(* PLC project Practical Work One, Rexroth ctrlX PLC Engineering ctrlX PLC 1.16.1, author Cedric Lenoir *)
(* stored: creationDateTime 2024-05-24T15:21:21.1871668, version 0.0, modificationDateTime 2024-05-24T15:19:54.2132771, organization HEVS *)
(* First Test for Practical Work One *)

TYPE UA_DigitalInput_32 : STRUCT
  Input_0_0 : BOOL;
  Input_0_1 : BOOL;
  Input_0_2 : BOOL;
  Input_0_3 : BOOL;
  Input_0_4 : BOOL;
  Input_0_5 : BOOL;
  Input_0_6 : BOOL;
  Input_0_7 : BOOL;
  Input_1_0 : BOOL;
  Input_1_1 : BOOL;
  Input_1_2 : BOOL;
  Input_1_3 : BOOL;
  Input_1_4 : BOOL;
  Input_1_5 : BOOL;
  Input_1_6 : BOOL;
  Input_1_7 : BOOL;
  Input_2_0 : BOOL;
  Input_2_1 : BOOL;
  Input_2_2 : BOOL;
  Input_2_3 : BOOL;
  Input_2_4 : BOOL;
  Input_2_5 : BOOL;
  Input_2_6 : BOOL;
  Input_2_7 : BOOL;
  Input_3_0 : BOOL;
  Input_3_1 : BOOL;
  Input_3_2 : BOOL;
  Input_3_3 : BOOL;
  Input_3_4 : BOOL;
  Input_3_5 : BOOL;
  Input_3_6 : BOOL;
  Input_3_7 : BOOL;
END_STRUCT;
END_TYPE

TYPE UA_DigitalOutput_32 : STRUCT
  Output_0_0 : BOOL;
  Output_0_1 : BOOL;
  Output_0_2 : BOOL;
  Output_0_3 : BOOL;
  Output_0_4 : BOOL;
  Output_0_5 : BOOL;
  Output_0_6 : BOOL;
  Output_0_7 : BOOL;
  Output_1_0 : BOOL;
  Output_1_1 : BOOL;
  Output_1_2 : BOOL;
  Output_1_3 : BOOL;
  Output_1_4 : BOOL;
  Output_1_5 : BOOL;
  Output_1_6 : BOOL;
  Output_1_7 : BOOL;
  Output_2_0 : BOOL;
  Output_2_1 : BOOL;
  Output_2_2 : BOOL;
  Output_2_3 : BOOL;
  Output_2_4 : BOOL;
  Output_2_5 : BOOL;
  Output_2_6 : BOOL;
  Output_2_7 : BOOL;
  Output_3_0 : BOOL;
  Output_3_1 : BOOL;
  Output_3_2 : BOOL;
  Output_3_3 : BOOL;
  Output_3_4 : BOOL;
  Output_3_5 : BOOL;
  Output_3_6 : BOOL;
  Output_3_7 : BOOL;
END_STRUCT;
END_TYPE

TYPE UA_ButtonAndSignal : STRUCT
  In_Estop : BOOL;
  In_Reset : BOOL;
  In_Start : BOOL;
  In_Stop : BOOL;
  Out_Idle : BOOL;
  Out_Execute : BOOL;
  Out_Stopped : BOOL;
END_STRUCT;
END_TYPE

TYPE UA_O300_DL : STRUCT
  Value : WORD;
  BCD1 : BOOL;
  Q : BOOL;
  A : BOOL;
END_STRUCT;
END_TYPE

TYPE UA_O300_ZL : STRUCT
  BCD1 : BOOL;
  Q : BOOL;
  A : BOOL;
END_STRUCT;
END_TYPE

TYPE UA_U300_D50 : STRUCT
  Value : DWORD;
  Scale : SINT;
  SSC1 : BOOL;
  SSC2 : BOOL;
  Q : BOOL;
  A : BOOL;
  SSC4 : BOOL;
END_STRUCT;
END_TYPE

(* www.hevs.ch Institut Systemes Industriels Project: Projet No: PW Move Absolute Author: Cedric Lenoir Date: 2023 October 16 Summary: List of commands for MoveAbsolute *)
TYPE ST_PlcOpenFbs : STRUCT
  bEnableRemote : BOOL;  (* If TRUE, the FB are driven manually from the HMI *)
  bEnableReadStatus : BOOL;
  bEnableReadPosition : BOOL;
  bEnableReadVelocity : BOOL;
  bMoveAbs : BOOL;
  bStop : BOOL;
  bPowerOn : BOOL;
  bReset : BOOL;
  strGetAxisStatus : STRING;  (* From arAxisStatus_gb[1].Data.PLCopenState; Exist in Data Layer too, s=motion/axs/Axis_X/state/opstate/plcopen *)
END_STRUCT;
END_TYPE

TYPE UA_U300_P50 : STRUCT
  Value : DWORD;
  Scale : SINT;
  SSC1 : BOOL;
  SSC2 : BOOL;
  Q : BOOL;
  A : BOOL;
  SSC4 : BOOL;
END_STRUCT;
END_TYPE

TYPE UA_Schunk_mms : STRUCT
  Value : WORD;
END_STRUCT;
END_TYPE

TYPE UA_Balluf_bcm0002 : STRUCT
  Data_1 : REAL;
  Data_2 : REAL;
  Data_3 : REAL;
  Temperature : REAL;
  Status : DWORD;
END_STRUCT;
END_TYPE

TYPE UA_Festo : STRUCT
  SetOut : BOOL;
END_STRUCT;
END_TYPE

TYPE UA_AnalogIn : STRUCT
  IW_04 : WORD;
  IW_06 : WORD;
  IW_08 : WORD;
  IW_10 : WORD;
  IW_12 : WORD;
  IW_14 : WORD;
  IW_16 : WORD;
  IW_18 : WORD;
END_STRUCT;
END_TYPE

TYPE UA_AnalogOut : STRUCT
  QW_04 : WORD;
  QW_06 : WORD;
  QW_08 : WORD;
  QW_10 : WORD;
END_STRUCT;
END_TYPE

TYPE UA_AboxInterface : STRUCT
  uaButtonAndSignal : UA_ButtonAndSignal;
  uaAnalogIn : UA_AnalogIn;
  uaAnalogOut : UA_AnalogOut;
  uaDigitalIn : UA_DigitalInput_32;
  uaDigitalOut : UA_DigitalOutput_32;
  uaO300_DL_Optic : UA_O300_DL;
  uaO300_ZL_Optic : UA_O300_ZL;
  uaU300_D50_Sound : UA_U300_D50;
  uaU300_P50_Sound : UA_U300_P50;
  uaSchunk : UA_Schunk_mms;
  uaSchunkGripper : UA_Festo;
  uaAccelerometer : UA_Balluf_bcm0002;
END_STRUCT;
END_TYPE

(* www.hevs.ch Institut Systemes Industriels Project: Projet No: PW Move Absolute Author: Cedric Lenoir Date: 2023 October 16 Summary: List of dynamic parameters for Move Absolute *)
TYPE ST_SetMotionParam : STRUCT
  rPosition_mm : LREAL;
  rVeloctiy_mm_s : LREAL;
  rAcceleration_mm_s2 : LREAL;
  rDeceleration_mm_s2 : LREAL;
  rJerk_mm_s3 : LREAL;
END_STRUCT;
END_TYPE

(* www.hevs.ch Institut Systemes Industriels Project: Projet No: PW Move Absolute Author: Cedric Lenoir Date: 2023 October 16 Summary: State Machine Info *)
TYPE ST_StateMachineInfo : STRUCT
  diState : DINT;
  eState : E_ExecuteCornerP5;
  strState : STRING;
END_STRUCT;
END_TYPE

{attribute 'qualified_only'}
{attribute 'strict'}
TYPE E_PackStates : (NotActive := 999, Aborted := 10, Clearing := 20, Stopped := 30, Resetting := 40, Idle := 50, Starting := 60, Stopping := 70, Aborting := 80, Execute := 90, Holding := 100, Held := 110, Unholding := 120, Suspending := 200, Suspended := 210, Unsuspending := 220, Completing := 300, Complete := 310) DINT;
END_TYPE

TYPE ST_PackState : STRUCT
  Aborted : BOOL;
  Clearing : BOOL;
  Stopped : BOOL;
  Resetting : BOOL;
  Idle : BOOL;
  Starting : BOOL;
  Stopping : BOOL;
  Aborting : BOOL;
  Execute : BOOL;
  Holding : BOOL;  (* Held Loop *)
  Held : BOOL;
  Unholding : BOOL;
  Suspending : BOOL;  (* Suspended Loop *)
  Suspended : BOOL;
  Unsuspending : BOOL;
  Completing : BOOL;  (* Complete Loop *)
  Complete : BOOL;
END_STRUCT;
END_TYPE

{attribute 'qualified_only'}
{attribute 'strict'}
TYPE E_Clearing : (eIdle := 99, eX_ErrorStop := 110, eX_Disabled := 120, eX_Enabled := 130, eY_ErrorStop := 210, eY_Disabled := 220, eY_Enabled := 230, eZ_ErrorStop := 310, eZ_Disabled := 320, eZ_Enabled := 330);
END_TYPE

{attribute 'qualified_only'}
{attribute 'strict'}
TYPE E_Stopping : (Idle := 99);
END_TYPE

{attribute 'qualified_only'}
{attribute 'strict'}
TYPE E_Resetting : (Idle := 99, eGripperSetOpen := 10, eGripperIsOpen := 20, eMotionInit_Z := 110, eMotionInitDone_Z := 120);
END_TYPE

{attribute 'qualified_only'}
{attribute 'strict'}
TYPE E_Starting : (Idle := 99, eMotionStarting := 10, eMotionStartingDone := 20);
END_TYPE

{attribute 'qualified_only'}
{attribute 'strict'}
TYPE E_InOpGripper : (IsIdle := 999, IsOpen := 10, IsClosed := 20, PartPresent := 30);
END_TYPE

TYPE ST_TestFbGripperHmi : STRUCT
  executeOpenDone : BOOL;
  executeCloseDone : BOOL;
  gripperStateClosed : BOOL;
  gripperStateOpen : BOOL;
  gripperStatePartPresent : BOOL;
  gripperStateError : BOOL;
  gripperStateInOp : BOOL;
END_STRUCT;
END_TYPE

{attribute 'qualified_only'}
{attribute 'strict'}
TYPE E_Aborting : (Idle := 99, Disabled := 1, ErrorStop := 2);
END_TYPE

TYPE ST_RemoteCyclicSetPosition : STRUCT
  in : ST_RemoteCyclicSetPositionIn;  (* Commands for program *)
  out : ST_RemoteCyclicSetPositionOut;  (* Status for program *)
END_STRUCT;
END_TYPE

TYPE ST_RemoteCyclicSetPositionIn : STRUCT
  lrStartPosition : LREAL := 0;  (* Set start position / Start of profile position *)
  lrEndPosition : LREAL := 50;  (* Set end position / End of profile position *)
  udiCycleTimeMultiplier : UDINT := 1000;  (* Cycle Time Multiplier, default is 1000 for 1000 ms *)
  bActivateCoupling : BOOL;  (* Activate coupling, when TRUE, axis position is set by fbGenerateProfile with 5th order polynomial *)
  bStartForward : BOOL;  (* Start polynomial profile forward *)
  lrProfileSetPosition : LREAL;  (* Set Position from Profile generator *)
END_STRUCT;
END_TYPE

TYPE ST_RemoteCyclicSetPositionOut : STRUCT
  bInitDone : BOOL;  (* Init done, ready for cyclic motion *)
  bError : BOOL;  (* There is an error *)
  bFwdDone : BOOL;  (* End of cyclic profile Forward *)
END_STRUCT;
END_TYPE

TYPE ST_Corner : STRUCT
  X : ST_SetMotionParam;
  Y : ST_SetMotionParam;
  Z : ST_SetMotionParam;
END_STRUCT;
END_TYPE

{attribute 'qualified_only'}
{attribute 'strict'}
TYPE E_InOperationDoneBase : (Idle := 999, Init := 10, InOp := 20, Error := 30, Done := 40);
END_TYPE

{attribute 'qualified_only'}
{attribute 'strict'}
TYPE E_ExecuteDone : (Idle := 999, Init := 10, InOp := 20, Done := 30, Error := 40);
END_TYPE

{attribute 'qualified_only'}
{attribute 'strict'}
TYPE E_InOperationBase : (Idle := 999, Init := 10, InOp := 20, Error := 30);
END_TYPE

{attribute 'qualified_only'}
{attribute 'strict'}
TYPE E_SubActiveP5 : (StartPointOut := 999, Running := 10, EndOfProfile := 20);
END_TYPE

(* www.hevs.ch Institut Systemes Industriels Project: Projet No: PW Move Absolute Author: Cedric Lenoir Date: 2024 April 02 Summary: Template of a program using PLCopen on partial Pack State Use a Cyclic Setpoint for motion in Pack Execute. *)
PROGRAM PRG_CyclicSetPoint
  VAR
    fbGripperState : FB_GripperState;  (* ********************************************************************************************************************* YOUR VARIABLES HERE ********************************************************************************************************************* *)
    fbOpenGripper : FB_OpenGripper;
    fbCloseGripper : FB_CloseGripper;
    uliCount : ULINT;
    bInitDone : BOOL;
    fbPackStates : FB_PackStates;  (* Pack Partial state machine *)
    eAborting : E_Aborting;
    eClearing : E_Clearing;
    eResetting : E_Resetting;
    eStarting : E_Starting;
    eStopping : E_Stopping;
    stStateMachineInfo : ST_StateMachineInfo;  (* State machine info for Execute *)
    stPlcOpenFbs : ST_PlcOpenFbs;  (* List of Structures *)
    stSetParam_X : ST_SetMotionParam := (rVeloctiy_mm_s := 2000, rAcceleration_mm_s2 := 1000, rDeceleration_mm_s2 := 1000, rJerk_mm_s3 := 1);
    stSetParam_Z : ST_SetMotionParam := (rVeloctiy_mm_s := 2000, rAcceleration_mm_s2 := 1000, rDeceleration_mm_s2 := 1000, rJerk_mm_s3 := 1);
    stCornerOne : ST_Corner := (X := (rVeloctiy_mm_s := 2000, rAcceleration_mm_s2 := 1000, rDeceleration_mm_s2 := 1000, rJerk_mm_s3 := 1), Y := (rVeloctiy_mm_s := 2000, rAcceleration_mm_s2 := 1000, rDeceleration_mm_s2 := 1000, rJerk_mm_s3 := 1), Z := (rVeloctiy_mm_s := 2000, rAcceleration_mm_s2 := 1000, rDeceleration_mm_s2 := 1000, rJerk_mm_s3 := 1));
    stCornerTwo : ST_Corner := (X := (rPosition_mm := 50, rVeloctiy_mm_s := 2000, rAcceleration_mm_s2 := 1000, rDeceleration_mm_s2 := 1000, rJerk_mm_s3 := 1), Y := (rVeloctiy_mm_s := 2000, rAcceleration_mm_s2 := 1000, rDeceleration_mm_s2 := 1000, rJerk_mm_s3 := 1), Z := (rVeloctiy_mm_s := 2000, rAcceleration_mm_s2 := 1000, rDeceleration_mm_s2 := 1000, rJerk_mm_s3 := 1));
    mcReadActualPos_X : MC_ReadActualPosition;  (* List of Function Blocks *)
    mcReadStatus_X : MC_ReadStatus;
    mcPower_X : MC_Power;
    mcMoveAbs_X : MC_MoveAbsolute;
    mcStop_X : MC_Stop := (Deceleration := 1);
    mcReset_X : MC_Reset;
    fbGenerateProfile : FB_GenerateP5;  (* Second part of variables are used to generate a motion profile using 5th order polynomial. Details of polynomials can be experimented using a mlx Matlab file. *)
    mcCyclicSetPoint : MB_CyclicSetPoint;
    mcReadActualPos_Z : MC_ReadActualPosition;  (* Simply used to move Z axis Up in a secure position *)
    mcReadStatus_Z : MC_ReadStatus;
    mcPower_Z : MC_Power;
    mcMoveAbs_Z : MC_MoveAbsolute;
    mcStop_Z : MC_Stop := (Deceleration := 1);
    mcReset_Z : MC_Reset;
    stTestFbGripperHmi : ST_TestFbGripperHmi;  (* Check your FB on HMI *)
  END_VAR

                    ACT_BaseInit();


IF fbPackStates.state.Execute THEN
	fbPackStates.Execute_SC := FALSE;
	(*
		Execute State Machine.
	*)
	CASE stStateMachineInfo.eState OF
		E_ExecuteCornerP5.eIdle :
			stStateMachineInfo.strState := 'Idle';
			
			stSetParam_X.rPosition_mm := 0;
			stStateMachineInfo.eState := E_ExecuteCornerP5.eMoveToCornerOne;

		E_ExecuteCornerP5.eMoveToCornerOne :
			stStateMachineInfo.strState := 'Motion To Corner One';
			IF mcMoveAbs_X.Done THEN
				stStateMachineInfo.eState := E_ExecuteCornerP5.eMoveToCornerOneDone; 
			END_IF

		E_ExecuteCornerP5.eMoveToCornerOneDone :
			stStateMachineInfo.strState := 'Motion To Corner One Done';
			// Corner 2 is like Corner three
			stSetParam_X.rPosition_mm := stCornerTwo.X.rPosition_mm;
			// stStateMachineInfo.eState := E_ExecuteCornerP5.eMoveToCornerThree;
			IF fbGripperState.IsOpen THEN
				stStateMachineInfo.eState := E_ExecuteCornerP5.eMoveToCornerTwo;
			END_IF;
			
 		(* Motion with P5*)   
    	E_ExecuteCornerP5.eMoveToCornerTwo :
			stStateMachineInfo.strState := 'Motion To Corner Two with P5';
			// Reset P5 to actual position
			// GVL_CyclSetPoint.stRemote.in.lrStartPosition := mcReadActualPos_X.Position;
			// Start position should be THIS position
			GVL_CyclSetPoint.stRemote.in.lrEndPosition := mcReadActualPos_X.Position;
			stStateMachineInfo.eState := E_ExecuteCornerP5.eEnableP5;
			
		E_ExecuteCornerP5.eEnableP5 :
			stStateMachineInfo.strState := 'Enable / Reset P5';
			IF fbGenerateProfile.Done THEN
				stStateMachineInfo.eState := E_ExecuteCornerP5.eCyclicSetPoint;
				;
			END_IF
		
		E_ExecuteCornerP5.eCyclicSetPoint :
			stStateMachineInfo.strState := 'Set Cyclic Set Point';
			IF mcCyclicSetPoint.Active THEN
				GVL_CyclSetPoint.stRemote.in.lrStartPosition := mcReadActualPos_X.Position;
				GVL_CyclSetPoint.stRemote.in.lrEndPosition := stCornerTwo.X.rPosition_mm;
				stStateMachineInfo.eState := E_ExecuteCornerP5.eFollowP5;
			END_IF
		
		E_ExecuteCornerP5.eFollowP5 :
			stStateMachineInfo.strState := 'Follow P5';
			IF fbGenerateProfile.Done THEN
				stStateMachineInfo.eState := E_ExecuteCornerP5.eStopCyclic;
			END_IF
		
		E_ExecuteCornerP5.eStopCyclic :
			stStateMachineInfo.strState := 'Stop Cyclic';
			IF mcStop_X.Done THEN
				stStateMachineInfo.eState := E_ExecuteCornerP5.eStopDone;
			END_IF
		
		E_ExecuteCornerP5.eStopDone :
			stStateMachineInfo.strState := 'Stop Done';
			stStateMachineInfo.eState := E_ExecuteCornerP5.eMoveToCornerTwoDone;	
		
		E_ExecuteCornerP5.eMoveToCornerTwoDone :			
			stStateMachineInfo.strState := 'Move to Corner Two Done';
			// Return to One.
			stSetParam_X.rPosition_mm := stCornerOne.X.rPosition_mm;
			IF fbGripperState.IsClosed THEN
				stStateMachineInfo.eState := E_ExecuteCornerP5.eMoveToCornerOne;
			END_IF; 

		E_ExecuteCornerP5.eMoveToCornerThree :
			stStateMachineInfo.strState := 'Motion to Corner Three';
			IF mcMoveAbs_X.Done THEN
				stStateMachineInfo.eState := E_ExecuteCornerP5.eMoveToCornerThreeDone; 
			END_IF

		E_ExecuteCornerP5.eMoveToCornerThreeDone :
			stStateMachineInfo.strState := 'Motion to Corner Three Done'; 

			stSetParam_X.rPosition_mm := 0;
			stStateMachineInfo.eState := E_ExecuteCornerP5.eMoveToCornerOne;

	END_CASE
	;
ELSE
	stStateMachineInfo.strState := 'Idle';
	stStateMachineInfo.eState := E_ExecuteCornerP5.eIdle;
END_IF

(*
	Try with 
*)
mcCyclicSetPoint.Execute := (GVL_CyclSetPoint.stRemote.in.bActivateCoupling AND stPlcOpenFbs.bEnableRemote) OR
	                        (stStateMachineInfo.eState = E_ExecuteCornerP5.eCyclicSetPoint);
mcCyclicSetPoint.SetPoint := GVL_CyclSetPoint.stRemote.in.lrProfileSetPosition;
mcCyclicSetPoint(Axis := GVL_AxisDefines.X_Axis);

(*
    Call FB at the end of the Program
*)
fbGenerateProfile(Enable := fbPackStates.state.Execute,
				  StartForward := (GVL_CyclSetPoint.stRemote.in.bStartForward AND stPlcOpenFbs.bEnableRemote) OR
                                   (stStateMachineInfo.eState = E_ExecuteCornerP5.eEnableP5)                   OR
                                   (stStateMachineInfo.eState = E_ExecuteCornerP5.eFollowP5),
                  startPosition_mm := GVL_CyclSetPoint.stRemote.in.lrStartPosition,		   // Start to try with 0
                  endPosition_mm := GVL_CyclSetPoint.stRemote.in.lrEndPosition,			   // Start to try with 50	
                  udiCyclTime_ms := GVL_CyclSetPoint.MOTION_CYCLE_TIME_ms,
                  udiCycleTimeMult := GVL_CyclSetPoint.stRemote.in.udiCycleTimeMultiplier, // Could be a parameter latter when all is working
                  arGoToPos := GVL_CyclSetPoint.arGoToPosition,
                  lrSetPosition => GVL_CyclSetPoint.stRemote.in.lrProfileSetPosition,
                  Done => GVL_CyclSetPoint.stRemote.out.bFwdDone);

(**********************************************************************************************************************
    Get Execute state machine in a DINT format
**********************************************************************************************************************)
stStateMachineInfo.diState := stStateMachineInfo.eState;
	
(**********************************************************************************************************************
	Utility FBs for motion, Do not modify
**********************************************************************************************************************)
ACT_ForAxis_X();
// Action for Y axis if defined
ACT_ForAxis_Z();

ACT_ForGripper();
                  

ACTION ACT_ForAxis_X:
                        (**********************************************************************************************************************
	X Axis
**********************************************************************************************************************)
mcReadStatus_X(Axis := GVL_AxisDefines.X_Axis,
               Enable := stPlcOpenFbs.bEnableReadStatus);

mcReadActualPos_X(Axis := GVL_AxisDefines.X_Axis,
                  Enable := stPlcOpenFbs.bEnableReadPosition);

mcPower_X(Axis := GVL_AxisDefines.X_Axis,
        Enable := (stPlcOpenFbs.bPowerOn AND stPlcOpenFbs.bEnableRemote) OR
                   		NOT stPlcOpenFbs.bEnableRemote AND 
				   		NOT (fbPackStates.state.Aborting OR
                             fbPackStates.state.Aborted));

mcStop_X(Axis := GVL_AxisDefines.X_Axis,
         Execute := (stPlcOpenFbs.bStop AND stPlcOpenFbs.bEnableRemote) OR
                    (fbPackStates.state.Stopping)                       OR
                    (stStateMachineInfo.eState = E_ExecuteCornerP5.eStopCyclic));

mcReset_X(Axis := GVL_AxisDefines.X_Axis,
        Execute := (stPlcOpenFbs.bReset AND stPlcOpenFbs.bEnableRemote) OR
                    fbPackStates.state.Aborting);

mcMoveAbs_X(Axis := GVL_AxisDefines.X_Axis,
            Position := stSetParam_X.rPosition_mm,
            Velocity := stSetParam_X.rVeloctiy_mm_s,
            Acceleration := stSetParam_X.rAcceleration_mm_s2,
            Deceleration := stSetParam_X.rDeceleration_mm_s2,
            Jerk := stSetParam_X.rJerk_mm_s3,
            Execute := (stPlcOpenFbs.bMoveAbs AND stPlcOpenFbs.bEnableRemote)    	OR
					   (eStarting = E_Starting.eMotionStarting)                  	OR
                       (stStateMachineInfo.eState = E_ExecuteCornerP5.eMoveToCornerOne)	OR              
                       (stStateMachineInfo.eState = E_ExecuteCornerP5.eMoveToCornerThree));  
						  

                      
END_ACTION

ACTION ACT_ForAxis_Z:
                        (**********************************************************************************************************************
	Z Axis
**********************************************************************************************************************)
mcReadStatus_Z(Axis := GVL_AxisDefines.Z_Axis,
               Enable := stPlcOpenFbs.bEnableReadStatus);

mcReadActualPos_Z(Axis := GVL_AxisDefines.Z_Axis,
                  Enable := stPlcOpenFbs.bEnableReadPosition);

mcPower_Z(Axis := GVL_AxisDefines.Z_Axis,
        Enable := (stPlcOpenFbs.bPowerOn AND stPlcOpenFbs.bEnableRemote) OR
                   		NOT stPlcOpenFbs.bEnableRemote AND 
				   		NOT (fbPackStates.state.Aborting OR
                             fbPackStates.state.Aborted));

// Note that a stop without deceleration leads to an error!!
mcStop_Z(Axis := GVL_AxisDefines.Z_Axis,
         Execute := (stPlcOpenFbs.bStop AND stPlcOpenFbs.bEnableRemote) OR
                     fbPackStates.state.Stopping);

mcReset_Z(Axis := GVL_AxisDefines.Z_Axis,
         Execute := (stPlcOpenFbs.bReset AND stPlcOpenFbs.bEnableRemote) OR
                     fbPackStates.state.Aborting);
					 
mcMoveAbs_Z(Axis := GVL_AxisDefines.Z_Axis,
            Position := stSetParam_Z.rPosition_mm,
            Velocity := stSetParam_Z.rVeloctiy_mm_s,
            Acceleration := stSetParam_Z.rAcceleration_mm_s2,
            Deceleration := stSetParam_Z.rDeceleration_mm_s2,
            Jerk := stSetParam_Z.rJerk_mm_s3,
            Execute := (stPlcOpenFbs.bMoveAbs AND stPlcOpenFbs.bEnableRemote)    OR
                       (eResetting = E_Resetting.eMotionInit_Z));  
                      
END_ACTION

ACTION ACT_BaseInit:
                        (*
    Some inits independant of the Main State Machine
*)
IF NOT bInitDone THEN
	bInitDone := TRUE;
    stPlcOpenFbs.bEnableReadStatus := TRUE;
    stPlcOpenFbs.bEnableReadPosition := TRUE;
    stPlcOpenFbs.bEnableReadVelocity := TRUE;
	// Init values to compile them and send to OPC_UA
	stTestFbGripperHmi.gripperStateClosed := FALSE;
	stTestFbGripperHmi.gripperStateOpen := FALSE;
	stTestFbGripperHmi.gripperStatePartPresent := FALSE;
	stTestFbGripperHmi.gripperStateError := FALSE;
	stTestFbGripperHmi.gripperStateInOp := FALSE;
	stTestFbGripperHmi.executeOpenDone := FALSE;
	stTestFbGripperHmi.executeCloseDone := FALSE;
END_IF

(*
    Remote conditions
*)
IF stPlcOpenFbs.bEnableRemote THEN
    IF mcMoveAbs_X.Done THEN
        stPlcOpenFbs.bMoveAbs := FALSE;
    END_IF
    IF mcStop_X.Done THEN
        stPlcOpenFbs.bStop := FALSE;
        stPlcOpenFbs.bMoveAbs := FALSE;
    END_IF
END_IF

// If remote, pack states are disabled
fbPackStates.SoftEstop := mcReadStatus_X.ErrorStop;
fbPackStates(Enable := NOT stPlcOpenFbs.bEnableRemote,
			 remote := GVL_Abox.uaAboxInterface.uaButtonAndSignal);
			 
(*
	Basically, only Acting state are used, wait state are doing nothing
	But sometimes, we could need to do something.. see Aborted.
*)

IF fbPackStates.state.Aborting THEN
	fbPackStates.Aborting_SC := TRUE;
ELSE
	;
END_IF

IF fbPackStates.state.Clearing THEN
	CASE eClearing OF
	E_Clearing.eIdle :
		IF mcReadStatus_X.Standstill THEN
			eClearing := E_Clearing.eY_ErrorStop;
		ELSIF mcReadStatus_X.ErrorStop THEN
			eClearing := E_Clearing.eX_ErrorStop;
		ELSE
			eClearing := E_Clearing.eX_Disabled;
		END_IF
	
	E_Clearing.eX_ErrorStop :
		IF mcReadStatus_X.Standstill THEN
			eClearing := E_Clearing.eY_ErrorStop;
		ELSE
			eClearing := E_Clearing.eX_Disabled;
		END_IF
	
	E_Clearing.eX_Disabled  :
		IF mcReadStatus_X.Standstill THEN
			eClearing := E_Clearing.eY_ErrorStop;
		ELSIF mcReadStatus_X.ErrorStop THEN
			eClearing := E_Clearing.eX_ErrorStop;
		END_IF
	
	E_Clearing.eX_Enabled   :
		IF mcReadStatus_X.Standstill THEN
			eClearing := E_Clearing.eY_ErrorStop;
		ELSIF mcReadStatus_X.ErrorStop THEN
			eClearing := E_Clearing.eX_ErrorStop;
		ELSE
			eClearing := E_Clearing.eX_Disabled;
		END_IF	

	E_Clearing.eY_ErrorStop :
		// No Y axis
		eClearing := E_Clearing.eZ_ErrorStop;
	
	E_Clearing.eY_Disabled  :
		eClearing := E_Clearing.eZ_ErrorStop;
	
	E_Clearing.eY_Enabled   :
		eClearing := E_Clearing.eZ_ErrorStop;

	E_Clearing.eZ_ErrorStop :
		IF mcReadStatus_Z.Standstill THEN
			eClearing := E_Clearing.eZ_Enabled;
		ELSE
			eClearing := E_Clearing.eZ_Disabled;
		END_IF	
	
	E_Clearing.eZ_Disabled  :
		IF mcReadStatus_Z.Standstill THEN
			eClearing := E_Clearing.eZ_Enabled;
		ELSIF mcReadStatus_Z.ErrorStop THEN
			eClearing := E_Clearing.eZ_ErrorStop;
		END_IF
	
	E_Clearing.eZ_Enabled   :;
		
	END_CASE
	// Reset Gripper in case fbOpenGripper and fbCloseGripper not presentz
	// GripperIsOpen   := TRUE;
	// GripperIsClosed	:= TRUE;	
	IF (eClearing = E_Clearing.eZ_Enabled) THEN
		fbPackStates.Clearing_SC := TRUE;
	ELSE
		fbPackStates.Clearing_SC := FALSE;
	END_IF
ELSE
	eClearing := E_Clearing.eIdle;
END_IF

IF fbPackStates.state.Stopping THEN
	IF mcReadStatus_X.Standstill AND
       mcReadStatus_Z.Standstill THEN
		fbPackStates.Stopping_SC := TRUE;
	ELSE
		fbPackStates.Stopping_SC := FALSE;
	END_IF
ELSE
	;
END_IF

(**********************************************************************************************************************
    Resetting
**********************************************************************************************************************)
IF fbPackStates.state.Resetting THEN
	fbPackStates.Resetting_SC := FALSE;
	CASE eResetting OF
		E_Resetting.Idle :
            stSetParam_Z.rPosition_mm := 0;
			stSetParam_Z.rVeloctiy_mm_s := 2000;  
			eResetting := E_Resetting.eGripperSetOpen;
			
		E_Resetting.eGripperSetOpen :
			IF fbGripperState.IsOpen THEN
				eResetting := E_Resetting.eGripperIsOpen;
			END_IF
			
		E_Resetting.eGripperIsOpen :
			// No Condition
			eResetting := E_Resetting.eMotionInit_Z;			
			
		E_Resetting.eMotionInit_Z :
			IF mcMoveAbs_Z.Done THEN
				eResetting := E_Resetting.eMotionInitDone_Z; 
			END_IF

		E_Resetting.eMotionInitDone_Z :
			;;
	END_CASE
	 
	IF eResetting = E_Resetting.eMotionInitDone_Z THEN
		fbPackStates.Resetting_SC := TRUE;
	END_IF
ELSE
	eResetting := E_Resetting.Idle;
END_IF

(**********************************************************************************************************************
    Starting
**********************************************************************************************************************)
IF fbPackStates.state.Starting THEN
	fbPackStates.Starting_SC := FALSE;
	CASE eStarting OF
		E_Starting.Idle :
			// Starting at corner Two
            stSetParam_X.rPosition_mm := stCornerOne.X.rPosition_mm;
			stSetParam_X.rVeloctiy_mm_s := stCornerOne.X.rVeloctiy_mm_s;  
			eStarting := E_Starting.eMotionStarting;

		E_Starting.eMotionStarting :
			IF mcMoveAbs_X.Done THEN
				eStarting := E_Starting.eMotionStartingDone; 
			END_IF

		E_Starting.eMotionStartingDone :
			;
						
	END_CASE
	 
	IF (eStarting = E_Starting.eMotionStartingDone) THEN
		fbPackStates.Starting_SC := TRUE;
	END_IF
ELSE
	eStarting := E_Starting.Idle;
END_IF
                      
END_ACTION

ACTION ACT_ForGripper:
                        fbGripperState.Enable := (stPlcOpenFbs.bEnableRemote)        		OR
                   		 (NOT stPlcOpenFbs.bEnableRemote 		AND 
				   		  NOT (fbPackStates.state.Aborting OR
                               fbPackStates.state.Aborted)); 
fbGripperState(hw := GVL_Abox.uaAboxInterface.uaSchunk);

stTestFbGripperHmi.gripperStateClosed := fbGripperState.IsClosed;
stTestFbGripperHmi.gripperStateOpen := fbGripperState.IsOpen;
stTestFbGripperHmi.gripperStatePartPresent := fbGripperState.PartPresent;
stTestFbGripperHmi.gripperStateError := fbGripperState.Error;
stTestFbGripperHmi.gripperStateInOp := fbGripperState.InOperation;

fbOpenGripper.Execute := (stStateMachineInfo.eState = E_ExecuteCornerP5.eMoveToCornerOneDone) OR 
                         (eResetting = E_Resetting.eGripperSetOpen);

fbCloseGripper.Execute := (stStateMachineInfo.eState = E_ExecuteCornerP5.eMoveToCornerTwoDone);

fbOpenGripper(hwEV := GVL_Abox.uaAboxInterface.uaSchunkGripper,
	          hwSensor := GVL_Abox.uaAboxInterface.uaSchunk,
			  Done => stTestFbGripperHmi.executeOpenDone);
			  
fbCloseGripper(hwEV := GVL_Abox.uaAboxInterface.uaSchunkGripper,
	          hwSensor := GVL_Abox.uaAboxInterface.uaSchunk,
			  Done => stTestFbGripperHmi.executeCloseDone);
                      
END_ACTION
END_PROGRAM

PROGRAM PRG_MapBox
  VAR
    UA_ReadCounterFromStation : DINT;  (* Write from Siemens to ctrX Core Used to check if read is running *)
    UA_ButtonAndSignal_In_Estop : BOOL;
    UA_ButtonAndSignal_In_Reset : BOOL;
    UA_ButtonAndSignal_In_Start : BOOL;
    UA_ButtonAndSignal_In_Stop : BOOL;
    UA_Balluf_bcm0002_Data_1 : REAL;
    UA_Balluf_bcm0002_Data_2 : REAL;
    UA_Balluf_bcm0002_Data_3 : REAL;
    UA_Balluf_bcm0002_Temperature : REAL;
    UA_Balluf_bcm0002_Status : DWORD;
    UA_Festo_SetOut : BOOL;
    UA_O300_DL_Value : WORD;
    UA_O300_DL_BCD1 : BOOL;
    UA_O300_DL_Q : BOOL;
    UA_O300_DL_A : BOOL;
    UA_O300_ZL_BCD1 : BOOL;
    UA_O300_ZL_Q : BOOL;
    UA_O300_ZL_A : BOOL;
    UA_U300_D50_Value : DWORD;
    UA_U300_D50_Scale : SINT;
    UA_U300_D50_SSC1 : BOOL;
    UA_U300_D50_SSC2 : BOOL;
    UA_U300_D50_Q : BOOL;
    UA_U300_D50_A : BOOL;
    UA_U300_D50_SSC4 : BOOL;
    UA_U300_P50_Value : DWORD;
    UA_U300_P50_Scale : SINT;
    UA_U300_P50_SSC1 : BOOL;
    UA_U300_P50_SSC2 : BOOL;
    UA_U300_P50_Q : BOOL;
    UA_U300_P50_A : BOOL;
    UA_U300_P50_SSC4 : BOOL;
    UA_DigitalInput_32_Input_0_0 : BOOL;
    UA_DigitalInput_32_Input_0_1 : BOOL;
    UA_DigitalInput_32_Input_0_2 : BOOL;
    UA_DigitalInput_32_Input_0_3 : BOOL;
    UA_DigitalInput_32_Input_0_4 : BOOL;
    UA_DigitalInput_32_Input_0_5 : BOOL;
    UA_DigitalInput_32_Input_0_6 : BOOL;
    UA_DigitalInput_32_Input_0_7 : BOOL;
    UA_DigitalInput_32_Input_1_0 : BOOL;
    UA_DigitalInput_32_Input_1_1 : BOOL;
    UA_DigitalInput_32_Input_1_2 : BOOL;
    UA_DigitalInput_32_Input_1_3 : BOOL;
    UA_DigitalInput_32_Input_1_4 : BOOL;
    UA_DigitalInput_32_Input_1_5 : BOOL;
    UA_DigitalInput_32_Input_1_6 : BOOL;
    UA_DigitalInput_32_Input_1_7 : BOOL;
    UA_DigitalInput_32_Input_2_0 : BOOL;
    UA_DigitalInput_32_Input_2_1 : BOOL;
    UA_DigitalInput_32_Input_2_2 : BOOL;
    UA_DigitalInput_32_Input_2_3 : BOOL;
    UA_DigitalInput_32_Input_2_4 : BOOL;
    UA_DigitalInput_32_Input_2_5 : BOOL;
    UA_DigitalInput_32_Input_2_6 : BOOL;
    UA_DigitalInput_32_Input_2_7 : BOOL;
    UA_DigitalInput_32_Input_3_0 : BOOL;
    UA_DigitalInput_32_Input_3_1 : BOOL;
    UA_DigitalInput_32_Input_3_2 : BOOL;
    UA_DigitalInput_32_Input_3_3 : BOOL;
    UA_DigitalInput_32_Input_3_4 : BOOL;
    UA_DigitalInput_32_Input_3_5 : BOOL;
    UA_DigitalInput_32_Input_3_6 : BOOL;
    UA_DigitalInput_32_Input_3_7 : BOOL;
    UA_WriteCounterToStation : DINT;  (* Siemens Read from ctrX Core Used to check if write is running *)
    UA_ButtonAndSignal_Out_Idle : BOOL;
    UA_ButtonAndSignal_Out_Execute : BOOL;
    UA_ButtonAndSignal_Out_Stopped : BOOL;
    UA_Schunk_mms_Value : WORD;
    UA_DigitalOutput_32_Output_0_0 : BOOL;
    UA_DigitalOutput_32_Output_0_1 : BOOL;
    UA_DigitalOutput_32_Output_0_2 : BOOL;
    UA_DigitalOutput_32_Output_0_3 : BOOL;
    UA_DigitalOutput_32_Output_0_4 : BOOL;
    UA_DigitalOutput_32_Output_0_5 : BOOL;
    UA_DigitalOutput_32_Output_0_6 : BOOL;
    UA_DigitalOutput_32_Output_0_7 : BOOL;
    UA_DigitalOutput_32_Output_1_0 : BOOL;
    UA_DigitalOutput_32_Output_1_1 : BOOL;
    UA_DigitalOutput_32_Output_1_2 : BOOL;
    UA_DigitalOutput_32_Output_1_3 : BOOL;
    UA_DigitalOutput_32_Output_1_4 : BOOL;
    UA_DigitalOutput_32_Output_1_5 : BOOL;
    UA_DigitalOutput_32_Output_1_6 : BOOL;
    UA_DigitalOutput_32_Output_1_7 : BOOL;
    UA_DigitalOutput_32_Output_2_0 : BOOL;
    UA_DigitalOutput_32_Output_2_1 : BOOL;
    UA_DigitalOutput_32_Output_2_2 : BOOL;
    UA_DigitalOutput_32_Output_2_3 : BOOL;
    UA_DigitalOutput_32_Output_2_4 : BOOL;
    UA_DigitalOutput_32_Output_2_5 : BOOL;
    UA_DigitalOutput_32_Output_2_6 : BOOL;
    UA_DigitalOutput_32_Output_2_7 : BOOL;
    UA_DigitalOutput_32_Output_3_0 : BOOL;
    UA_DigitalOutput_32_Output_3_1 : BOOL;
    UA_DigitalOutput_32_Output_3_2 : BOOL;
    UA_DigitalOutput_32_Output_3_3 : BOOL;
    UA_DigitalOutput_32_Output_3_4 : BOOL;
    UA_DigitalOutput_32_Output_3_5 : BOOL;
    UA_DigitalOutput_32_Output_3_6 : BOOL;
    UA_DigitalOutput_32_Output_3_7 : BOOL;
  END_VAR

                        (*
        Values from Profinet Station
    *)
    
    // Get Value from Profinet Station with UA Client Write
	GVL_Abox.uaAboxInterface.uaButtonAndSignal.In_Estop     := UA_ButtonAndSignal_In_Estop;
	GVL_Abox.uaAboxInterface.uaButtonAndSignal.In_Reset     := UA_ButtonAndSignal_In_Reset;
	GVL_Abox.uaAboxInterface.uaButtonAndSignal.In_Start     := UA_ButtonAndSignal_In_Start;
	GVL_Abox.uaAboxInterface.uaButtonAndSignal.In_Stop      := UA_ButtonAndSignal_In_Stop;
    // Values from Balluff accelerometer
    GVL_Abox.uaAboxInterface.uaAccelerometer.Data_1         := UA_Balluf_bcm0002_Data_1;
    GVL_Abox.uaAboxInterface.uaAccelerometer.Data_2         := UA_Balluf_bcm0002_Data_1;
    GVL_Abox.uaAboxInterface.uaAccelerometer.Data_3         := UA_Balluf_bcm0002_Data_1;
    GVL_Abox.uaAboxInterface.uaAccelerometer.Status         := UA_Balluf_bcm0002_Status;
    GVL_Abox.uaAboxInterface.uaAccelerometer.Temperature    := UA_Balluf_bcm0002_Temperature;

    // Values from Baumer O300 DL
    GVL_Abox.uaAboxInterface.uaO300_DL_Optic.Value          := UA_O300_DL_Value;                
    GVL_Abox.uaAboxInterface.uaO300_DL_Optic.A              := UA_O300_DL_A;                
    GVL_Abox.uaAboxInterface.uaO300_DL_Optic.Q              := UA_O300_DL_Q;                
    GVL_Abox.uaAboxInterface.uaO300_DL_Optic.BCD1           := UA_O300_DL_BCD1;                

    // Values from Baumer O300 ZL                
    GVL_Abox.uaAboxInterface.uaO300_ZL_Optic.A              := UA_O300_ZL_A;                
    GVL_Abox.uaAboxInterface.uaO300_ZL_Optic.Q              := UA_O300_ZL_Q;                
    GVL_Abox.uaAboxInterface.uaO300_ZL_Optic.BCD1           := UA_O300_ZL_BCD1;                

    // Values from Baumer U300 D50
    GVL_Abox.uaAboxInterface.uaU300_D50_Sound.Value         := UA_U300_D50_Value;  
    GVL_Abox.uaAboxInterface.uaU300_D50_Sound.A             := UA_U300_D50_A;  
    GVL_Abox.uaAboxInterface.uaU300_D50_Sound.Q             := UA_U300_D50_Q;  
    GVL_Abox.uaAboxInterface.uaU300_D50_Sound.Scale         := UA_U300_D50_Scale;  
    GVL_Abox.uaAboxInterface.uaU300_D50_Sound.SSC1          := UA_U300_D50_SSC1;  
    GVL_Abox.uaAboxInterface.uaU300_D50_Sound.SSC2          := UA_U300_D50_SSC2;  
    GVL_Abox.uaAboxInterface.uaU300_D50_Sound.SSC4          := UA_U300_D50_SSC4;  
    
    // Values from Baumer U300 P50
    GVL_Abox.uaAboxInterface.uaU300_P50_Sound.Value         := UA_U300_P50_Value;  
    GVL_Abox.uaAboxInterface.uaU300_P50_Sound.A             := UA_U300_P50_A;  
    GVL_Abox.uaAboxInterface.uaU300_P50_Sound.Q             := UA_U300_P50_Q;  
    GVL_Abox.uaAboxInterface.uaU300_P50_Sound.Scale         := UA_U300_P50_Scale;  
    GVL_Abox.uaAboxInterface.uaU300_P50_Sound.SSC1          := UA_U300_P50_SSC1;  
    GVL_Abox.uaAboxInterface.uaU300_P50_Sound.SSC2          := UA_U300_P50_SSC2;  
    GVL_Abox.uaAboxInterface.uaU300_P50_Sound.SSC4          := UA_U300_P50_SSC4;  
    
    // Values from Gripper sensor
    GVL_Abox.uaAboxInterface.uaSchunk.Value                 := UA_Schunk_mms_Value;  
    
    // Get 32 Digital Input
    GVL_Abox.uaAboxInterface.uaDigitalIn.Input_0_0          := UA_DigitalInput_32_Input_0_0;
    GVL_Abox.uaAboxInterface.uaDigitalIn.Input_0_1          := UA_DigitalInput_32_Input_0_1;
    GVL_Abox.uaAboxInterface.uaDigitalIn.Input_0_2          := UA_DigitalInput_32_Input_0_2;
    GVL_Abox.uaAboxInterface.uaDigitalIn.Input_0_3          := UA_DigitalInput_32_Input_0_3;
    GVL_Abox.uaAboxInterface.uaDigitalIn.Input_0_4          := UA_DigitalInput_32_Input_0_4;
    GVL_Abox.uaAboxInterface.uaDigitalIn.Input_0_5          := UA_DigitalInput_32_Input_0_5;
    GVL_Abox.uaAboxInterface.uaDigitalIn.Input_0_6          := UA_DigitalInput_32_Input_0_6;
    GVL_Abox.uaAboxInterface.uaDigitalIn.Input_0_7          := UA_DigitalInput_32_Input_0_7;
    GVL_Abox.uaAboxInterface.uaDigitalIn.Input_1_0          := UA_DigitalInput_32_Input_1_0;
    GVL_Abox.uaAboxInterface.uaDigitalIn.Input_1_1          := UA_DigitalInput_32_Input_1_1;
    GVL_Abox.uaAboxInterface.uaDigitalIn.Input_1_2          := UA_DigitalInput_32_Input_1_2;
    GVL_Abox.uaAboxInterface.uaDigitalIn.Input_1_3          := UA_DigitalInput_32_Input_1_3;
    GVL_Abox.uaAboxInterface.uaDigitalIn.Input_1_4          := UA_DigitalInput_32_Input_1_4;
    GVL_Abox.uaAboxInterface.uaDigitalIn.Input_1_5          := UA_DigitalInput_32_Input_1_5;
    GVL_Abox.uaAboxInterface.uaDigitalIn.Input_1_6          := UA_DigitalInput_32_Input_1_6;
    GVL_Abox.uaAboxInterface.uaDigitalIn.Input_1_7          := UA_DigitalInput_32_Input_1_7;
    GVL_Abox.uaAboxInterface.uaDigitalIn.Input_2_0          := UA_DigitalInput_32_Input_2_0;
    GVL_Abox.uaAboxInterface.uaDigitalIn.Input_2_1          := UA_DigitalInput_32_Input_2_1;
    GVL_Abox.uaAboxInterface.uaDigitalIn.Input_2_2          := UA_DigitalInput_32_Input_2_2;
    GVL_Abox.uaAboxInterface.uaDigitalIn.Input_2_3          := UA_DigitalInput_32_Input_2_3;
    GVL_Abox.uaAboxInterface.uaDigitalIn.Input_2_4          := UA_DigitalInput_32_Input_2_4;
    GVL_Abox.uaAboxInterface.uaDigitalIn.Input_2_5          := UA_DigitalInput_32_Input_2_5;
    GVL_Abox.uaAboxInterface.uaDigitalIn.Input_2_6          := UA_DigitalInput_32_Input_2_6;
    GVL_Abox.uaAboxInterface.uaDigitalIn.Input_2_7          := UA_DigitalInput_32_Input_2_7;
    GVL_Abox.uaAboxInterface.uaDigitalIn.Input_3_0          := UA_DigitalInput_32_Input_3_0;
    GVL_Abox.uaAboxInterface.uaDigitalIn.Input_3_1          := UA_DigitalInput_32_Input_3_1;
    GVL_Abox.uaAboxInterface.uaDigitalIn.Input_3_2          := UA_DigitalInput_32_Input_3_2;
    GVL_Abox.uaAboxInterface.uaDigitalIn.Input_3_3          := UA_DigitalInput_32_Input_3_3;
    GVL_Abox.uaAboxInterface.uaDigitalIn.Input_3_4          := UA_DigitalInput_32_Input_3_4;
    GVL_Abox.uaAboxInterface.uaDigitalIn.Input_3_5          := UA_DigitalInput_32_Input_3_5;
    GVL_Abox.uaAboxInterface.uaDigitalIn.Input_3_6          := UA_DigitalInput_32_Input_3_6;
    GVL_Abox.uaAboxInterface.uaDigitalIn.Input_3_7          := UA_DigitalInput_32_Input_3_7;
    
    (*
        Values to Profinet Station
    *)
	UA_WriteCounterToStation := UA_WriteCounterToStation + 1;

    // Set Visual Signals
	UA_ButtonAndSignal_Out_Execute 	:= GVL_Abox.uaAboxInterface.uaButtonAndSignal.Out_Execute;
	UA_ButtonAndSignal_Out_Idle 	:= GVL_Abox.uaAboxInterface.uaButtonAndSignal.Out_Idle;
	UA_ButtonAndSignal_Out_Stopped	:= GVL_Abox.uaAboxInterface.uaButtonAndSignal.Out_Stopped;
    
    // Set Gripper value
    UA_Festo_SetOut                 := NOT GVL_Abox.uaAboxInterface.uaSchunkGripper.SetOut;
    
    // Set 32 digital outputs
    UA_DigitalOutput_32_Output_0_0  := GVL_Abox.uaAboxInterface.uaDigitalOut.Output_0_0;
    UA_DigitalOutput_32_Output_0_1  := GVL_Abox.uaAboxInterface.uaDigitalOut.Output_0_1;
    UA_DigitalOutput_32_Output_0_2  := GVL_Abox.uaAboxInterface.uaDigitalOut.Output_0_2;
    UA_DigitalOutput_32_Output_0_3  := GVL_Abox.uaAboxInterface.uaDigitalOut.Output_0_3;
    UA_DigitalOutput_32_Output_0_4  := GVL_Abox.uaAboxInterface.uaDigitalOut.Output_0_4;
    UA_DigitalOutput_32_Output_0_5  := GVL_Abox.uaAboxInterface.uaDigitalOut.Output_0_5;
    UA_DigitalOutput_32_Output_0_6  := GVL_Abox.uaAboxInterface.uaDigitalOut.Output_0_6;
    UA_DigitalOutput_32_Output_0_7  := GVL_Abox.uaAboxInterface.uaDigitalOut.Output_0_7;
    UA_DigitalOutput_32_Output_1_0  := GVL_Abox.uaAboxInterface.uaDigitalOut.Output_1_0;
    UA_DigitalOutput_32_Output_1_1  := GVL_Abox.uaAboxInterface.uaDigitalOut.Output_1_1;
    UA_DigitalOutput_32_Output_1_2  := GVL_Abox.uaAboxInterface.uaDigitalOut.Output_1_2;
    UA_DigitalOutput_32_Output_1_3  := GVL_Abox.uaAboxInterface.uaDigitalOut.Output_1_3;
    UA_DigitalOutput_32_Output_1_4  := GVL_Abox.uaAboxInterface.uaDigitalOut.Output_1_4;
    UA_DigitalOutput_32_Output_1_5  := GVL_Abox.uaAboxInterface.uaDigitalOut.Output_1_5;
    UA_DigitalOutput_32_Output_1_6  := GVL_Abox.uaAboxInterface.uaDigitalOut.Output_1_6;
    UA_DigitalOutput_32_Output_1_7  := GVL_Abox.uaAboxInterface.uaDigitalOut.Output_1_7;
    UA_DigitalOutput_32_Output_2_0  := GVL_Abox.uaAboxInterface.uaDigitalOut.Output_2_0;
    UA_DigitalOutput_32_Output_2_1  := GVL_Abox.uaAboxInterface.uaDigitalOut.Output_2_1;
    UA_DigitalOutput_32_Output_2_2  := GVL_Abox.uaAboxInterface.uaDigitalOut.Output_2_2;
    UA_DigitalOutput_32_Output_2_3  := GVL_Abox.uaAboxInterface.uaDigitalOut.Output_2_3;
    UA_DigitalOutput_32_Output_2_4  := GVL_Abox.uaAboxInterface.uaDigitalOut.Output_2_4;
    UA_DigitalOutput_32_Output_2_5  := GVL_Abox.uaAboxInterface.uaDigitalOut.Output_2_5;
    UA_DigitalOutput_32_Output_2_6  := GVL_Abox.uaAboxInterface.uaDigitalOut.Output_2_6;
    UA_DigitalOutput_32_Output_2_7  := GVL_Abox.uaAboxInterface.uaDigitalOut.Output_2_7;
    UA_DigitalOutput_32_Output_3_0  := GVL_Abox.uaAboxInterface.uaDigitalOut.Output_3_0;
    UA_DigitalOutput_32_Output_3_1  := GVL_Abox.uaAboxInterface.uaDigitalOut.Output_3_1;
    UA_DigitalOutput_32_Output_3_2  := GVL_Abox.uaAboxInterface.uaDigitalOut.Output_3_2;
    UA_DigitalOutput_32_Output_3_3  := GVL_Abox.uaAboxInterface.uaDigitalOut.Output_3_3;
    UA_DigitalOutput_32_Output_3_4  := GVL_Abox.uaAboxInterface.uaDigitalOut.Output_3_4;
    UA_DigitalOutput_32_Output_3_5  := GVL_Abox.uaAboxInterface.uaDigitalOut.Output_3_5;
    UA_DigitalOutput_32_Output_3_6  := GVL_Abox.uaAboxInterface.uaDigitalOut.Output_3_6;
    UA_DigitalOutput_32_Output_3_7  := GVL_Abox.uaAboxInterface.uaDigitalOut.Output_3_7;
    
PRG_CHECK_IO();
                  
END_PROGRAM

PROGRAM PRG_CHECK_IO
  VAR
    testButton_1 : BOOL;
    testButton_2 : BOOL;
    testButton_3 : BOOL;
    clignote : TON;
    changeMeSlow : BOOL;
    clignoteSlow : TON;
    changeMe : BOOL;
    NotResetTest : BOOL := TRUE;
  END_VAR

                    testButton_1 := GVL_Abox.uaAboxInterface.uaButtonAndSignal.In_Reset;
testButton_2 := GVL_Abox.uaAboxInterface.uaButtonAndSignal.In_Start;
testButton_3 := GVL_Abox.uaAboxInterface.uaButtonAndSignal.In_Stop;

IF GVL_Abox.uaAboxInterface.uaButtonAndSignal.In_Reset AND
   NotResetTest										   THEN
	NotResetTest := FALSE;
	
    GVL_Abox.uaAboxInterface.uaSchunkGripper.SetOut := FALSE;
    
    GVL_Abox.uaAboxInterface.uaButtonAndSignal.Out_Execute := FALSE;	
    GVL_Abox.uaAboxInterface.uaButtonAndSignal.Out_Idle := FALSE;	
    GVL_Abox.uaAboxInterface.uaButtonAndSignal.Out_Stopped := FALSE;	

    GVL_Abox.uaAboxInterface.uaDigitalOut.Output_0_0 := FALSE;
    GVL_Abox.uaAboxInterface.uaDigitalOut.Output_0_1 := FALSE;
    GVL_Abox.uaAboxInterface.uaDigitalOut.Output_0_2 := FALSE;
    GVL_Abox.uaAboxInterface.uaDigitalOut.Output_0_3 := FALSE;
    GVL_Abox.uaAboxInterface.uaDigitalOut.Output_0_4 := FALSE;
    GVL_Abox.uaAboxInterface.uaDigitalOut.Output_0_5 := FALSE;
    GVL_Abox.uaAboxInterface.uaDigitalOut.Output_0_6 := FALSE;
    GVL_Abox.uaAboxInterface.uaDigitalOut.Output_0_7 := FALSE;
    
    GVL_Abox.uaAboxInterface.uaDigitalOut.Output_1_0 := FALSE;
    GVL_Abox.uaAboxInterface.uaDigitalOut.Output_1_1 := FALSE;
    GVL_Abox.uaAboxInterface.uaDigitalOut.Output_1_2 := FALSE;
    GVL_Abox.uaAboxInterface.uaDigitalOut.Output_1_3 := FALSE;
    GVL_Abox.uaAboxInterface.uaDigitalOut.Output_1_4 := FALSE;
    GVL_Abox.uaAboxInterface.uaDigitalOut.Output_1_5 := FALSE;
    GVL_Abox.uaAboxInterface.uaDigitalOut.Output_1_6 := FALSE;
    GVL_Abox.uaAboxInterface.uaDigitalOut.Output_1_7 := FALSE;
    
    GVL_Abox.uaAboxInterface.uaDigitalOut.Output_2_0 := FALSE;
    GVL_Abox.uaAboxInterface.uaDigitalOut.Output_2_1 := FALSE;
    GVL_Abox.uaAboxInterface.uaDigitalOut.Output_2_2 := FALSE;
    GVL_Abox.uaAboxInterface.uaDigitalOut.Output_2_3 := FALSE;
    GVL_Abox.uaAboxInterface.uaDigitalOut.Output_2_4 := FALSE;
    GVL_Abox.uaAboxInterface.uaDigitalOut.Output_2_5 := FALSE;
    GVL_Abox.uaAboxInterface.uaDigitalOut.Output_2_6 := FALSE;
    GVL_Abox.uaAboxInterface.uaDigitalOut.Output_2_7 := FALSE;

    GVL_Abox.uaAboxInterface.uaDigitalOut.Output_3_0 := FALSE;
    GVL_Abox.uaAboxInterface.uaDigitalOut.Output_3_1 := FALSE;
    GVL_Abox.uaAboxInterface.uaDigitalOut.Output_3_2 := FALSE;
    GVL_Abox.uaAboxInterface.uaDigitalOut.Output_3_3 := FALSE;
    GVL_Abox.uaAboxInterface.uaDigitalOut.Output_3_4 := FALSE;
    GVL_Abox.uaAboxInterface.uaDigitalOut.Output_3_5 := FALSE;
    GVL_Abox.uaAboxInterface.uaDigitalOut.Output_3_6 := FALSE;
    GVL_Abox.uaAboxInterface.uaDigitalOut.Output_3_7 := FALSE;	
END_IF

IF GVL_Abox.uaAboxInterface.uaButtonAndSignal.In_Reset AND
   GVL_Abox.uaAboxInterface.uaButtonAndSignal.In_Start AND
   GVL_Abox.uaAboxInterface.uaButtonAndSignal.In_Stop  THEN
	NotResetTest := TRUE;
END_IF


IF NotResetTest THEN 
	
	// Quick Blink
	clignote(IN := changeMe,
			 PT := T#500MS);
			 
	IF clignote.Q THEN
		changeMe := FALSE;
	ELSE
		changeMe := TRUE;
	END_IF

	// Slow Blink
	clignoteSlow(IN := changeMeSlow,
			 	 PT := T#2500MS);
			 
	IF clignoteSlow.Q THEN
		changeMeSlow := FALSE;
	ELSE
		changeMeSlow := TRUE;
	END_IF
	
	IF (NOT GVL_Abox.uaAboxInterface.uaSchunkGripper.SetOut) AND clignoteSlow.Q THEN
		GVL_Abox.uaAboxInterface.uaSchunkGripper.SetOut := TRUE;
	ELSIF GVL_Abox.uaAboxInterface.uaSchunkGripper.SetOut AND clignoteSlow.Q THEN
		GVL_Abox.uaAboxInterface.uaSchunkGripper.SetOut := FALSE;
	END_IF
	
	IF (NOT GVL_Abox.uaAboxInterface.uaDigitalOut.Output_0_0) AND clignote.Q THEN
		GVL_Abox.uaAboxInterface.uaButtonAndSignal.Out_Execute := TRUE;	
		GVL_Abox.uaAboxInterface.uaButtonAndSignal.Out_Idle := TRUE;	
		GVL_Abox.uaAboxInterface.uaButtonAndSignal.Out_Stopped := TRUE;	
	
		GVL_Abox.uaAboxInterface.uaDigitalOut.Output_0_0 := TRUE;
		GVL_Abox.uaAboxInterface.uaDigitalOut.Output_0_1 := TRUE;
		GVL_Abox.uaAboxInterface.uaDigitalOut.Output_0_2 := TRUE;
		GVL_Abox.uaAboxInterface.uaDigitalOut.Output_0_3 := TRUE;
		GVL_Abox.uaAboxInterface.uaDigitalOut.Output_0_4 := TRUE;
		GVL_Abox.uaAboxInterface.uaDigitalOut.Output_0_5 := TRUE;
		GVL_Abox.uaAboxInterface.uaDigitalOut.Output_0_6 := TRUE;
		GVL_Abox.uaAboxInterface.uaDigitalOut.Output_0_7 := TRUE;
		
		GVL_Abox.uaAboxInterface.uaDigitalOut.Output_1_0 := TRUE;
		GVL_Abox.uaAboxInterface.uaDigitalOut.Output_1_1 := TRUE;
		GVL_Abox.uaAboxInterface.uaDigitalOut.Output_1_2 := TRUE;
		GVL_Abox.uaAboxInterface.uaDigitalOut.Output_1_3 := TRUE;
		GVL_Abox.uaAboxInterface.uaDigitalOut.Output_1_4 := TRUE;
		GVL_Abox.uaAboxInterface.uaDigitalOut.Output_1_5 := TRUE;
		GVL_Abox.uaAboxInterface.uaDigitalOut.Output_1_6 := TRUE;
		GVL_Abox.uaAboxInterface.uaDigitalOut.Output_1_7 := TRUE;
		
		GVL_Abox.uaAboxInterface.uaDigitalOut.Output_2_0 := TRUE;
		GVL_Abox.uaAboxInterface.uaDigitalOut.Output_2_1 := TRUE;
		GVL_Abox.uaAboxInterface.uaDigitalOut.Output_2_2 := TRUE;
		GVL_Abox.uaAboxInterface.uaDigitalOut.Output_2_3 := TRUE;
		GVL_Abox.uaAboxInterface.uaDigitalOut.Output_2_4 := TRUE;
		GVL_Abox.uaAboxInterface.uaDigitalOut.Output_2_5 := TRUE;
		GVL_Abox.uaAboxInterface.uaDigitalOut.Output_2_6 := TRUE;
		GVL_Abox.uaAboxInterface.uaDigitalOut.Output_2_7 := TRUE;

		GVL_Abox.uaAboxInterface.uaDigitalOut.Output_3_0 := TRUE;
		GVL_Abox.uaAboxInterface.uaDigitalOut.Output_3_1 := TRUE;
		GVL_Abox.uaAboxInterface.uaDigitalOut.Output_3_2 := TRUE;
		GVL_Abox.uaAboxInterface.uaDigitalOut.Output_3_3 := TRUE;
		GVL_Abox.uaAboxInterface.uaDigitalOut.Output_3_4 := TRUE;
		GVL_Abox.uaAboxInterface.uaDigitalOut.Output_3_5 := TRUE;
		GVL_Abox.uaAboxInterface.uaDigitalOut.Output_3_6 := TRUE;
		GVL_Abox.uaAboxInterface.uaDigitalOut.Output_3_7 := TRUE;
	ELSIF GVL_Abox.uaAboxInterface.uaDigitalOut.Output_0_0 AND clignote.Q THEN
		GVL_Abox.uaAboxInterface.uaButtonAndSignal.Out_Execute := FALSE;	
		GVL_Abox.uaAboxInterface.uaButtonAndSignal.Out_Idle := FALSE;	
		GVL_Abox.uaAboxInterface.uaButtonAndSignal.Out_Stopped := FALSE;	

		GVL_Abox.uaAboxInterface.uaDigitalOut.Output_0_0 := FALSE;
		GVL_Abox.uaAboxInterface.uaDigitalOut.Output_0_1 := FALSE;
		GVL_Abox.uaAboxInterface.uaDigitalOut.Output_0_2 := FALSE;
		GVL_Abox.uaAboxInterface.uaDigitalOut.Output_0_3 := FALSE;
		GVL_Abox.uaAboxInterface.uaDigitalOut.Output_0_4 := FALSE;
		GVL_Abox.uaAboxInterface.uaDigitalOut.Output_0_5 := FALSE;
		GVL_Abox.uaAboxInterface.uaDigitalOut.Output_0_6 := FALSE;
		GVL_Abox.uaAboxInterface.uaDigitalOut.Output_0_7 := FALSE;
		
		GVL_Abox.uaAboxInterface.uaDigitalOut.Output_1_0 := FALSE;
		GVL_Abox.uaAboxInterface.uaDigitalOut.Output_1_1 := FALSE;
		GVL_Abox.uaAboxInterface.uaDigitalOut.Output_1_2 := FALSE;
		GVL_Abox.uaAboxInterface.uaDigitalOut.Output_1_3 := FALSE;
		GVL_Abox.uaAboxInterface.uaDigitalOut.Output_1_4 := FALSE;
		GVL_Abox.uaAboxInterface.uaDigitalOut.Output_1_5 := FALSE;
		GVL_Abox.uaAboxInterface.uaDigitalOut.Output_1_6 := FALSE;
		GVL_Abox.uaAboxInterface.uaDigitalOut.Output_1_7 := FALSE;
		
		GVL_Abox.uaAboxInterface.uaDigitalOut.Output_2_0 := FALSE;
		GVL_Abox.uaAboxInterface.uaDigitalOut.Output_2_1 := FALSE;
		GVL_Abox.uaAboxInterface.uaDigitalOut.Output_2_2 := FALSE;
		GVL_Abox.uaAboxInterface.uaDigitalOut.Output_2_3 := FALSE;
		GVL_Abox.uaAboxInterface.uaDigitalOut.Output_2_4 := FALSE;
		GVL_Abox.uaAboxInterface.uaDigitalOut.Output_2_5 := FALSE;
		GVL_Abox.uaAboxInterface.uaDigitalOut.Output_2_6 := FALSE;
		GVL_Abox.uaAboxInterface.uaDigitalOut.Output_2_7 := FALSE;

		GVL_Abox.uaAboxInterface.uaDigitalOut.Output_3_0 := FALSE;
		GVL_Abox.uaAboxInterface.uaDigitalOut.Output_3_1 := FALSE;
		GVL_Abox.uaAboxInterface.uaDigitalOut.Output_3_2 := FALSE;
		GVL_Abox.uaAboxInterface.uaDigitalOut.Output_3_3 := FALSE;
		GVL_Abox.uaAboxInterface.uaDigitalOut.Output_3_4 := FALSE;
		GVL_Abox.uaAboxInterface.uaDigitalOut.Output_3_5 := FALSE;
		GVL_Abox.uaAboxInterface.uaDigitalOut.Output_3_6 := FALSE;
		GVL_Abox.uaAboxInterface.uaDigitalOut.Output_3_7 := FALSE;
	END_IF;
END_IF
                  
END_PROGRAM

FUNCTION_BLOCK FB_PackStates
  VAR_INPUT
    Enable : BOOL;
    SoftEstop : BOOL;
    Hold : BOOL := FALSE;
    Unhold : BOOL := FALSE;
    Clearing_SC : BOOL := TRUE;
    Stopping_SC : BOOL := TRUE;
    Aborting_SC : BOOL := TRUE;
    Resetting_SC : BOOL := TRUE;
    Starting_SC : BOOL := TRUE;
    Execute_SC : BOOL := FALSE;
    Holding_SC : BOOL := FALSE;
    Unholding_SC : BOOL := FALSE;
  END_VAR
  VAR_IN_OUT
    remote : UA_ButtonAndSignal;
  END_VAR
  VAR_OUTPUT
    state : ST_PackState;
    strState : STRING;
  END_VAR
  VAR
    initialized : BOOL;
    ePackStates : E_PackStates;
    rTrigStop : R_TRIG;
    rTrigStart : R_TRIG;
    rTrigReset : R_TRIG;
    clignote : TON;
    changeMe : BOOL;
  END_VAR

                    // 
//	Init
//
IF Enable THEN
	IF NOT initialized THEN
		// Init at Aborted when entering state machine.
		initialized := TRUE;
		ePackStates := E_PackStates.Aborted;
	END_IF;
ELSE
	ePackStates := E_PackStates.NotActive;
	initialized := FALSE;
END_IF

//
//	Manage Inputs
//
rTrigStop(CLK := remote.In_Stop);
rTrigStart(CLK := remote.In_Start);
rTrigReset(CLK := remote.In_Reset);

CASE ePackStates OF
	E_PackStates.NotActive	:
		strState := 'Not Active';
		;
	E_PackStates.Aborting 	:;
		strState := 'Aborting';
		IF Aborting_SC THEN
			ePackStates := E_PackStates.Aborted;
		END_IF
		
	E_PackStates.Aborted 	:
		strState := 'Aborted';
		IF rTrigReset.Q THEN
			ePackStates := E_PackStates.Clearing;
		END_IF
	
	E_PackStates.Clearing 	:
		strState := 'Clearing';
		// E-Stop Active Low
		IF NOT remote.In_Estop OR SoftEstop THEN
			ePackStates := E_PackStates.Aborting;
		ELSIF Clearing_SC THEN
			ePackStates := E_PackStates.Stopped;	
		END_IF

	E_PackStates.Stopped 	:
		strState := 'Stopped';
		// E-Stop Active Low
		IF NOT remote.In_Estop OR SoftEstop THEN
			ePackStates := E_PackStates.Aborting;
		ELSIF rTrigReset.Q THEN
			ePackStates := E_PackStates.Resetting;
		END_IF

	E_PackStates.Stopping 	:
		strState := 'Stopping';
		// E-Stop Active Low
		IF NOT remote.In_Estop OR SoftEstop THEN
			ePackStates := E_PackStates.Aborting;
		ELSIF Stopping_SC THEN
			ePackStates := E_PackStates.Stopped;
		END_IF

	E_PackStates.Resetting 	:
		strState := 'Resetting';
		// E-Stop Active Low
		IF NOT remote.In_Estop OR SoftEstop THEN
			ePackStates := E_PackStates.Aborting;
		ELSIF rTrigStop.Q THEN
			ePackStates := E_PackStates.Stopping;
		ELSIF Resetting_SC THEN
			ePackStates := E_PackStates.Idle;			
		END_IF

	E_PackStates.Idle 		:
		strState := 'Idle';
		// E-Stop Active Low
		IF NOT remote.In_Estop OR SoftEstop THEN
			ePackStates := E_PackStates.Aborting;
		ELSIF rTrigStop.Q THEN
			ePackStates := E_PackStates.Stopping;
		ELSIF rTrigStart.Q THEN
			ePackStates := E_PackStates.Starting;
		END_IF

	E_PackStates.Starting 	:
		strState := 'Starting';
		// E-Stop Active Low
		IF NOT remote.In_Estop OR SoftEstop THEN
			ePackStates := E_PackStates.Aborting;
		ELSIF rTrigStop.Q THEN
			ePackStates := E_PackStates.Stopping;
		ELSIF Starting_SC THEN
			ePackStates := E_PackStates.Execute;	
		END_IF

	E_PackStates.Execute 	:
		strState := 'Execute';
		// E-Stop Active Low
		IF NOT remote.In_Estop OR SoftEstop THEN
			ePackStates := E_PackStates.Aborting;
		ELSIF rTrigStop.Q THEN
			ePackStates := E_PackStates.Stopping;
		ELSIF Hold		 THEN
			ePackStates := E_PackStates.Holding;	
		ELSIF Execute_SC THEN
			ePackStates := E_PackStates.Execute;	
		END_IF
		
	(* Held Loop *)
	E_PackStates.Holding	:;
		strState := 'Holding';
		// E-Stop Active Low
		IF NOT remote.In_Estop OR SoftEstop THEN
			ePackStates := E_PackStates.Aborting;
		ELSIF rTrigStop.Q THEN
			ePackStates := E_PackStates.Stopping;
		ELSIF Holding_SC THEN
			ePackStates := E_PackStates.Held;	
		END_IF
		
	E_PackStates.Held		:;
		strState := 'Held';
		// E-Stop Active Low
		IF NOT remote.In_Estop OR SoftEstop THEN
			ePackStates := E_PackStates.Aborting;
		ELSIF rTrigStop.Q THEN
			ePackStates := E_PackStates.Stopping;
		ELSIF Unhold THEN
			ePackStates := E_PackStates.Unholding;	
		END_IF

	E_PackStates.Unholding	:;
		strState := 'Unholding';
		// E-Stop Active Low
		IF NOT remote.In_Estop OR SoftEstop THEN
			ePackStates := E_PackStates.Aborting;
		ELSIF rTrigStop.Q THEN
			ePackStates := E_PackStates.Stopping;
		ELSIF Unholding_SC THEN
			ePackStates := E_PackStates.Execute;	
		END_IF

END_CASE

// Quick Blink
clignote(IN := changeMe,
		 PT := T#500MS);
			 
IF clignote.Q THEN
	changeMe := FALSE;
ELSE
	changeMe := TRUE;
END_IF

// Set Output states
state.Aborting	:= (ePackStates = E_PackStates.Aborting);
state.Aborted	:= (ePackStates = E_PackStates.Aborted);
state.Clearing	:= (ePackStates = E_PackStates.Clearing);
state.Stopped	:= (ePackStates = E_PackStates.Stopped);
state.Stopping	:= (ePackStates = E_PackStates.Stopping);
state.Resetting	:= (ePackStates = E_PackStates.Resetting);
state.Idle		:= (ePackStates = E_PackStates.Idle);
state.Starting	:= (ePackStates = E_PackStates.Starting);
state.Execute	:= (ePackStates = E_PackStates.Execute);

// Set Output signals
remote.Out_Stopped := (ePackStates = E_PackStates.Stopped);

IF ePackStates = E_PackStates.Starting THEN
	IF remote.Out_Execute AND clignote.Q THEN
		remote.Out_Execute := FALSE;
	ELSIF NOT remote.Out_Execute AND clignote.Q THEN
		remote.Out_Execute := TRUE;
	END_IF
ELSE
	remote.Out_Execute := (ePackStates = E_PackStates.Execute);	
END_IF

IF ePackStates = E_PackStates.Resetting THEN
	IF remote.Out_Idle AND clignote.Q THEN
		remote.Out_Idle := FALSE;
	ELSIF NOT remote.Out_Idle AND clignote.Q THEN
		remote.Out_Idle := TRUE;
	END_IF
ELSE
	remote.Out_Idle := (ePackStates = E_PackStates.Idle);	
END_IF

IF ePackStates = E_PackStates.Stopping OR 
   ePackStates = E_PackStates.Clearing THEN
	IF remote.Out_Stopped AND clignote.Q THEN
		remote.Out_Stopped := FALSE;
	ELSIF NOT remote.Out_Stopped AND clignote.Q THEN
		remote.Out_Stopped := TRUE;
	END_IF
ELSE
	remote.Out_Stopped := (ePackStates = E_PackStates.Stopped);	
END_IF
                  
END_FUNCTION_BLOCK

FUNCTION_BLOCK FB_GripperState
  VAR_INPUT
    Enable : BOOL;  (* Default Input *)
    thOpen : WORD := 50;  (* User Defined Inputs *)
    thClose : WORD := 950;
    thPartMin : WORD := 800;
    thPartMax : WORD := 860;
  END_VAR
  VAR_IN_OUT
    hw : UA_Schunk_mms;
  END_VAR
  VAR_OUTPUT
    InOperation : BOOL;  (* Default Outputs *)
    Error : BOOL;
    IsOpen : BOOL;  (* User Outputs *)
    IsClosed : BOOL;
    PartPresent : BOOL;
  END_VAR
  VAR
    eInOperationBase : E_InOperationBase := E_InOperationBase.Idle;
    eInOpGripper : E_InOpGripper := E_InOpGripper.IsIdle;
    tonIdleCondition : TON;
  END_VAR

                    (*
	Input management. While gripper is moving, it must not be seen as an Idle Condition
	Here we use a timer as Input Management.
*)

tonIdleCondition(IN := (((hw.Value > thOpen) AND (hw.Value < thPartMin))  OR
		                ((hw.Value < thClose) AND (hw.Value > thPartMax))),
				 PT := T#1S);

(*
	Main State Machine
*)
CASE eInOperationBase OF
	E_InOperationBase.Idle :
		IF Enable THEN
			eInOperationBase := E_InOperationBase.Init;	
		END_IF
		
	E_InOperationBase.Init :
		IF NOT Enable THEN
			eInOperationBase := E_InOperationBase.Idle;
		ELSIF tonIdleCondition.Q THEN
		    eInOpGripper := E_InOpGripper.IsIdle;
		 	eInOperationBase := E_InOperationBase.Error;
		ELSE // Init internal state machine and jump in it
			IF hw.Value < thOpen THEN
				eInOpGripper := E_InOpGripper.IsOpen;
			ELSIF hw.Value > thClose THEN
				eInOpGripper := E_InOpGripper.IsClosed;
			ELSE
				eInOpGripper := E_InOpGripper.PartPresent;
			END_IF
			eInOperationBase := E_InOperationBase.InOp;
		END_IF
		
	E_InOperationBase.InOp :
		(*
			Sub State Machine Here
		*)
		// Machine initilized in E_InOperationBase.Init
		// Error condition again, air pressure could be removed while machine is running
		IF NOT Enable THEN
			eInOperationBase := E_InOperationBase.Idle;
		ELSIF tonIdleCondition.Q THEN			// Error condition
		    eInOpGripper := E_InOpGripper.IsIdle;
		 	eInOperationBase := E_InOperationBase.Error;
		ELSE // Init internal state machine and jump in it
			CASE eInOpGripper OF
				E_InOpGripper.IsIdle :
					; // Do nothing, condition is checked in IF
				E_InOpGripper.IsOpen :
					IF hw.Value > thClose THEN
						eInOpGripper := E_InOpGripper.IsClosed;
					ELSIF (hw.Value > thPartMin) AND (hw.Value < thPartMax) THEN
						eInOpGripper := E_InOpGripper.PartPresent;
					END_IF
				E_InOpGripper.IsClosed :
					IF hw.Value < thOpen THEN
						eInOpGripper := E_InOpGripper.IsOpen;
					END_IF
				E_InOpGripper.PartPresent :
					IF hw.Value < thOpen THEN
						eInOpGripper := E_InOpGripper.IsOpen;
					END_IF
			END_CASE
		END_IF
	E_InOperationBase.Error :
		IF NOT Enable THEN
			eInOperationBase := E_InOperationBase.Idle;
		END_IF
END_CASE

(*
	Output Management
*)
InOperation			:= (eInOperationBase = E_InOperationBase.InOp);
Error				:= (eInOperationBase = E_InOperationBase.Error);

IsOpen				:= (eInOperationBase = E_InOperationBase.InOp) AND (eInOpGripper = E_InOpGripper.IsOpen);
IsClosed			:= (eInOperationBase = E_InOperationBase.InOp) AND (eInOpGripper = E_InOpGripper.IsClosed);
PartPresent			:= (eInOperationBase = E_InOperationBase.InOp) AND (eInOpGripper = E_InOpGripper.PartPresent);

                  
END_FUNCTION_BLOCK

FUNCTION_BLOCK FB_CloseGripper
  VAR_INPUT
    Execute : BOOL;
    thClosedMin : WORD := 950;
  END_VAR
  VAR_IN_OUT
    hwSensor : UA_Schunk_mms;
    hwEV : UA_Festo;
  END_VAR
  VAR_OUTPUT
    Done : BOOL;
    Active : BOOL;
    Error : BOOL;
  END_VAR
  VAR
    tnCheckDone : TON;
    rExecute : R_TRIG;
    eExecuteDone : E_ExecuteDone;
  END_VAR

                    (* 
	Manage Inputs
*)
rExecute(CLK := Execute);
// Timer.Q true if Execute and not threshold for more thant 1 sec.
tnCheckDone(IN := Execute AND NOT (hwSensor.Value > thClosedMin),
	        PT := T#1S);

CASE eExecuteDone OF
	E_ExecuteDone.Idle :
		IF rExecute.Q THEN
			eExecuteDone := E_ExecuteDone.Init;
		END_IF

	E_ExecuteDone.Init :
		// No init
		IF tnCheckDone.Q THEN
			eExecuteDone := E_ExecuteDone.Error;
		ELSE
			eExecuteDone := E_ExecuteDone.InOp;
		END_IF

	E_ExecuteDone.InOp :
		IF tnCheckDone.Q THEN
			eExecuteDone := E_ExecuteDone.Error;
		ELSIF (hwSensor.Value > thClosedMin) THEN
			eExecuteDone := E_ExecuteDone.Done;
		END_IF
	
	E_ExecuteDone.Done :
		IF NOT Execute THEN
			eExecuteDone := E_ExecuteDone.Idle;
		END_IF

	E_ExecuteDone.Error :
		IF NOT Execute THEN
			eExecuteDone := E_ExecuteDone.Idle;
		END_IF
END_CASE

IF eExecuteDone = E_ExecuteDone.InOp THEN
	hwEV.SetOut := FALSE;
END_IF

Done := (eExecuteDone = E_ExecuteDone.Done);
Active := (eExecuteDone = E_ExecuteDone.Init) OR (eExecuteDone = E_ExecuteDone.InOp) ;
Error := (eExecuteDone = E_ExecuteDone.Error);
                  
END_FUNCTION_BLOCK

FUNCTION_BLOCK FB_OpenGripper
  VAR_INPUT
    Execute : BOOL;
    thOpenMax : WORD := 50;
  END_VAR
  VAR_IN_OUT
    hwSensor : UA_Schunk_mms;
    hwEV : UA_Festo;
  END_VAR
  VAR_OUTPUT
    Done : BOOL;
    Active : BOOL;
    Error : BOOL;
  END_VAR
  VAR
    tnCheckDone : TON;
    rExecute : R_TRIG;
    eExecuteDone : E_ExecuteDone;
  END_VAR

                    (* 
	Manage Inputs
*)
rExecute(CLK := Execute);
// Timer.Q true if Execute and not threshold for more thant 1 sec.
tnCheckDone(IN := Execute AND NOT (hwSensor.Value < thOpenMax),
	        PT := T#1S);

CASE eExecuteDone OF
	E_ExecuteDone.Idle :
		IF rExecute.Q THEN
			eExecuteDone := E_ExecuteDone.Init;
		END_IF

	E_ExecuteDone.Init :
		// No init
		IF tnCheckDone.Q THEN
			eExecuteDone := E_ExecuteDone.Error;
		ELSE
			eExecuteDone := E_ExecuteDone.InOp;
		END_IF

	E_ExecuteDone.InOp :
		IF tnCheckDone.Q THEN
			eExecuteDone := E_ExecuteDone.Error;
		ELSIF (hwSensor.Value < thOpenMax) THEN
			eExecuteDone := E_ExecuteDone.Done;
		END_IF
	
	E_ExecuteDone.Done :
		IF NOT Execute THEN
			eExecuteDone := E_ExecuteDone.Idle;
		END_IF

	E_ExecuteDone.Error :
		IF NOT Execute THEN
			eExecuteDone := E_ExecuteDone.Idle;
		END_IF
END_CASE

IF eExecuteDone = E_ExecuteDone.InOp THEN
	hwEV.SetOut := TRUE;
END_IF

Done := (eExecuteDone = E_ExecuteDone.Done);
Active := (eExecuteDone = E_ExecuteDone.Init) OR (eExecuteDone = E_ExecuteDone.InOp) ;
Error := (eExecuteDone = E_ExecuteDone.Error);
                  
END_FUNCTION_BLOCK

FUNCTION_BLOCK FB_GenerateP5
  VAR_INPUT
    Enable : BOOL;  (* Std Inout for EnableDoneBase *)
    StartForward : BOOL;  (* Start of motion at rising edge. *)
    startPosition_mm : LREAL := 0;  (* Should be 0 for first version, could be extended for any position *)
    endPosition_mm : LREAL := 0;  (* Should be limited to 100 mm *)
    udiCyclTime_ms : UDINT;  (* Cycle time in ms of the task where FB is running. *)
    udiCycleTimeMult : UDINT;  (* Cycle time multiplier, used to compute duration of motion This could be made automatically later, Now result in Output Cycle Time Multiplier, default is 1000 for 1000 ms *)
  END_VAR
  VAR_IN_OUT
    arGoToPos : ARRAY[0..GVL_CyclSetPoint.c_uiMaxProfilePoints] OF LREAL;  (* Used for verification of data, we do not nead them for motion *)
  END_VAR
  VAR_OUTPUT
    Done : BOOL;  (* Motion finished *)
    Active : BOOL;  (* Point generator active *)
    Error : BOOL;
    udiMotionTime_ms : UDINT;  (* Is time to execute the profile in ms Multiplication of udiCyclTime_ms x udiCycleTimeMult *)
    lrSetPosition : LREAL;  (* Motion set position *)
  END_VAR
  VAR
    bErrorTimeMultToBig : BOOL;  (* True if udiCycleTimeMult Exceeds, FB not executed *)
    discreteTimeIndex : UDINT;  (* Time index of position *)
    lrTimeScaler : LREAL;  (* Ce machin là va devoir être expliqué avec pas mal de détail en théorie. *)
    eInOpeDoneBase : E_InOperationDoneBase;  (* Internal state machine *)
    eSubActiveP5 : E_SubActiveP5;
  END_VAR

                    CASE eInOpeDoneBase OF
	E_InOperationDoneBase.Idle 	:
		IF Enable THEN
			eInOpeDoneBase := E_InOperationDoneBase.Init; 
		END_IF

	E_InOperationDoneBase.Init 	:
		IF udiCycleTimeMult > GVL_CyclSetPoint.c_uiMaxProfilePoints THEN
			eInOpeDoneBase := E_InOperationDoneBase.Error;
		ELSIF Enable THEN
			// Hence this value cannot be modified while moving
			udiMotionTime_ms := udiCyclTime_ms * udiCycleTimeMult;
			eInOpeDoneBase := E_InOperationDoneBase.InOp;
			eSubActiveP5 := E_SubActiveP5.StartPointOut;
		ELSE
			eInOpeDoneBase := E_InOperationDoneBase.Idle;
		END_IF

	E_InOperationDoneBase.InOp 	:
		// No error condition
		IF Enable THEN
			CASE eSubActiveP5 OF
				E_SubActiveP5.StartPointOut :
					IF StartForward THEN
						lrSetPosition := startPosition_mm;
						discreteTimeIndex := 0; 
						lrTimeScaler := 1/UDINT_TO_LREAL(udiCycleTimeMult);
						eSubActiveP5 := E_SubActiveP5.Running;
					END_IF
					
				E_SubActiveP5.Running		:
					// Matlab operation with some modifications : 
					// position_yAxis(iLoop) = (t_xAxis(iLoop)^3 * P5_position(4) + t_xAxis(iLoop)^4 * P5_position(5) + t_xAxis(iLoop)^5 * P5_position(6)) * y_scaling_mm;
					arGoToPos[discreteTimeIndex] := startPosition_mm                                                 + 
													(EXPT(lrTimeScaler*discreteTimeIndex,3) * GVL_CyclSetPoint.P5[4] +
													 EXPT(lrTimeScaler*discreteTimeIndex,4) * GVL_CyclSetPoint.P5[5] +
													 EXPT(lrTimeScaler*discreteTimeIndex,5) * GVL_CyclSetPoint.P5[6]) * (endPosition_mm - startPosition_mm);
					// Set new value
					lrSetPosition := arGoToPos[discreteTimeIndex];
					// inc at each cycle
					discreteTimeIndex := discreteTimeIndex + 1;
					IF discreteTimeIndex > udiCycleTimeMult THEN
						eSubActiveP5 := E_SubActiveP5.EndOfProfile;
					END_IF // discreteTimeIndex > udiCycleTimeMult
	
					E_SubActiveP5.EndOfProfile  :
						;
	
					IF eSubActiveP5 = E_SubActiveP5.EndOfProfile THEN
						eInOpeDoneBase := E_InOperationDoneBase.Done;
					END_IF
			END_CASE 
		ELSE
			eInOpeDoneBase := E_InOperationDoneBase.Idle;
		END_IF // Enable
		
	E_InOperationDoneBase.Done	:
		IF NOT StartForward THEN
			eInOpeDoneBase := E_InOperationDoneBase.InOp;
			// reset internal state machine
			eSubActiveP5 := E_SubActiveP5.StartPointOut;
		END_IF

	E_InOperationDoneBase.Error :
		bErrorTimeMultToBig := TRUE;
		IF NOT Enable THEN
			bErrorTimeMultToBig := FALSE;
		END_IF
		
END_CASE

(*
	Manage outputs
*)
Active := (eInOpeDoneBase = E_InOperationDoneBase.InOp);
Done := (eInOpeDoneBase = E_InOperationDoneBase.Done);
Error := (eInOpeDoneBase = E_InOperationDoneBase.Error);


                  
END_FUNCTION_BLOCK

CONFIGURATION PracticalWork_07
  RESOURCE BaseInterfaceUa ON PLC
    {attribute 'qualified_only'}
    VAR_GLOBAL  (* GVL_Abox *)
      uaAboxInterface : UA_AboxInterface;
    END_VAR
    {attribute 'qualified_only'}
    VAR_GLOBAL  (* GVL_AxisDefines *)
      X_Axis : MB_AXISIF_REF := (AxisName := 'Axis_1', AxisNo := 1);
      Y_Axis : MB_AXISIF_REF := (AxisName := 'Axis_2', AxisNo := 2);
      Z_Axis : MB_AXISIF_REF := (AxisName := 'Axis_3', AxisNo := 3);
    END_VAR
    {attribute 'qualified_only'}
    VAR_GLOBAL  (* GVL_CyclSetPoint *)
      stRemote : ST_RemoteCyclicSetPosition := (in := (lrEndPosition := 50));  (* Remote for this program *)
      arGoToPosition : ARRAY[0..c_uiMaxProfilePoints] OF LREAL;  (* These values are for check only, it is possible to work without buffer *)
      c_uiMaxProfilePoints : UDINT := 1000;  (* 1001 points of 2 ms for max 2 [s] motion *)
      P5 : ARRAY[1..6] OF LREAL := [0, 0, 0, 10, -15, 6];  (* P5 Polynomial P5(0) to P5(5) exp 0 to 5 *)
      MOTION_CYCLE_TIME_ms : UDINT := 2;  (* equal to real time bus *)
    END_VAR
    TASK MainTask(PRIORITY := 30);
    PROGRAM PRG_CyclicSetPoint WITH MainTask : PRG_CyclicSetPoint;
    PROGRAM PRG_MapBox WITH MainTask : PRG_MapBox;
  END_RESOURCE
END_CONFIGURATION

CONFIGURATION Realtime_Data
END_CONFIGURATION
